FUNCTION proj0_TupleStruct_3: DINT
{ S7_Optimized_Access := 'true' }
    VAR_INPUT
        tuple: TupleStruct_3;
    END_VAR

BEGIN
    proj0_TupleStruct_3 := tuple.field0;
END_FUNCTION
